FUNCTION_BLOCK FILE_WRITER_7_LINEAR_MOVE (* Writes equation coeficients to a file (7 coef) for LINEAR_MOVE block *)
  (* Standard: 61499-2 *)
  (* Version 1.0, 23-03-12, GASR, Universidade do Estado de Santa Catarina *)
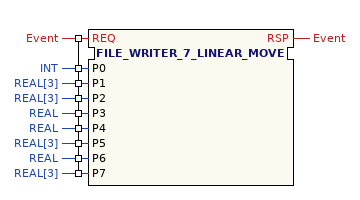
  EVENT_INPUT
    REQ WITH P0, P1, P2, P3, P4, P5, P6, P7; (* Request file storage *)
  END_EVENT
  EVENT_OUTPUT
    RSP; (* Finished operation *)
  END_EVENT
  VAR_INPUT
    P0 : INT; (* Process/equation id *)
    P1 : ARRAY [0..2] OF REAL; (* Coeficient 1 *)
    P2 : ARRAY [0..2] OF REAL; (* Coeficient 2 *)
    P3 : REAL; (* Coeficient 3 *)
    P4 : REAL; (* Coeficient 4 *)
    P5 : ARRAY [0..2] OF REAL; (* Coeficient 5 *)
    P6 : REAL; (* Coeficient 6 *)
    P7 : ARRAY [0..2] OF REAL; (* Coeficient 7 *)
  END_VAR
  SERVICE FILE_WRITER_7/MACHINE (* Coeficient file storage service *)
    SEQUENCE normal_establishment
      FILE_WRITER_7.REQ(P0,P1,P2,P3,P4,P5,P6,P7) -> MACHINE.write-file();
      MACHINE.response() -> FILE_WRITER_7.RSP();
    END_SEQUENCE
  END_SERVICE
END_FUNCTION_BLOCK
